Staubli VAL3: MessageHeader.pjx

--- MessageHeader.pjx ---
Parameters version=s7.7.2 stackSize=5000 millimeterUnit=true
Program file=start.pgx
Program file=stop.pgx
Data file=MessageHeader.dtx

--- MessageHeader.dtx ---
public num nMagicNumber
public num nProtocolVersion
public num nMsgType
public num nMsgSequenceNumber
public num nPayloadSize
public num nHeaderSize
